// TIA Portal V18 export
TYPE "SubAssemblyID_ShW"
// stored: IsFailsafeCompliant false
   STRUCT
      _1 : Struct
         "name" : String[48];
         code : String[48];
         number : DInt;
      END_STRUCT;
      _2 : Struct
         "name" : String[48];
         code : String[48];
         number : DInt;
      END_STRUCT;
      _3 : Struct
         "name" : String[48];
         code : String[48];
         number : DInt;
      END_STRUCT;
      _4 : Struct
         "name" : String[48];
         code : String[48];
         number : DInt;
      END_STRUCT;
      _5 : Struct
         "name" : String[48];
         code : String[48];
         number : DInt;
      END_STRUCT;
   END_STRUCT;
END_TYPE
